{attribute 'qualified_only'}
{attribute 'strict'}
TYPE E_ServoState :
(
	DEFAULT	  := -1,
	OFF		  := 0,
	DISABLED,
	FAULTED,
	ENABLED,
	STANDBY,
	HOMING,
	MOVE_ABS,
	MOVE_REL,
	MOVE_SCAN,
	INTERLOCK_MOTION
);
END_TYPE
//  DEFAULT = '-1'

(* stored: Version 1.1.0.1, ProductVersion 3.1.4024.12
   EnumerationTextList E_ServoState: Id {bb00bc6e-88fe-45b3-81de-794230a1e1bb} *)
